% RSLogix 500 project Examen Certificación.RSS, saved by version 9.00.00.04 %
PROJECT "UNTITLED"    % processor: MicroLogix 1200 %

PROGRAM FILES
  LAD 2 "MAIN"  6 rungs
  LAD 3 "ENTRADAS"  6 rungs
  LAD 4 "SALIDAS"  4 rungs
  LAD 5 "MANUAL"  4 rungs
  LAD 6 "AUTOMATICO"  11 rungs
  LAD 7 "PARPADEOS"  5 rungs
  LAD 8 "LS"  2 rungs

DATA FILES
  O0 OUTPUT  4 elements
  I1 INPUT  4 elements
  S2 STATUS  66 elements
  B3 BINARY  4 elements
  T4 TIMER  3 elements
  C5 COUNTER  2 elements
  R6 CONTROL  1 elements
  N7 INTEGER  1 elements
  F8 FLOAT  1 elements

LADDER 2 "MAIN"
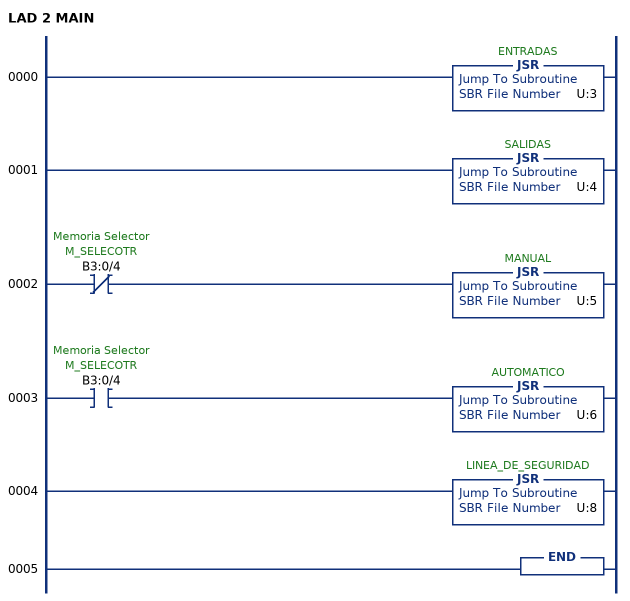
% Rung: 0 %
SOR JSR U:3 EOR
%   U:3  ENTRADAS %
% Rung: 1 %
SOR JSR U:4 EOR
%   U:4  SALIDAS %
% Rung: 2 %
SOR XIO B3:0/4 JSR U:5 EOR
%   B3:0/4  M_SELECOTR  "Memoria Selector" %
%   U:5  MANUAL %
% Rung: 3 %
SOR XIC B3:0/4 JSR U:6 EOR
%   B3:0/4  M_SELECOTR  "Memoria Selector" %
%   U:6  AUTOMATICO %
% Rung: 4 %
SOR JSR U:8 EOR
%   U:8  LINEA_DE_SEGURIDAD %
% Rung: 5 %
SOR END EOR

LADDER 3 "ENTRADAS"
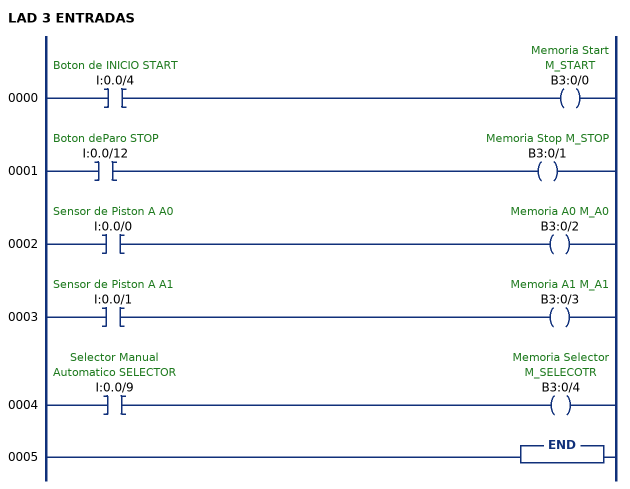
% Rung: 0 %
SOR XIC I:0.0/4 OTE B3:0/0 EOR
%   I:0.0/4  START  "Boton de INICIO" %
%   B3:0/0  M_START  "Memoria Start" %
% Rung: 1 %
SOR XIC I:0.0/12 OTE B3:0/1 EOR
%   I:0.0/12  STOP  "Boton deParo" %
%   B3:0/1  M_STOP  "Memoria Stop" %
% Rung: 2 %
SOR XIC I:0.0/0 OTE B3:0/2 EOR
%   I:0.0/0  A0  "Sensor de Piston A" %
%   B3:0/2  M_A0  "Memoria A0" %
% Rung: 3 %
SOR XIC I:0.0/1 OTE B3:0/3 EOR
%   I:0.0/1  A1  "Sensor de Piston A" %
%   B3:0/3  M_A1  "Memoria A1" %
% Rung: 4 %
SOR XIC I:0.0/9 OTE B3:0/4 EOR
%   I:0.0/9  SELECTOR  "Selector Manual Automatico" %
%   B3:0/4  M_SELECOTR  "Memoria Selector" %
% Rung: 5 %
SOR END EOR

LADDER 4 "SALIDAS"
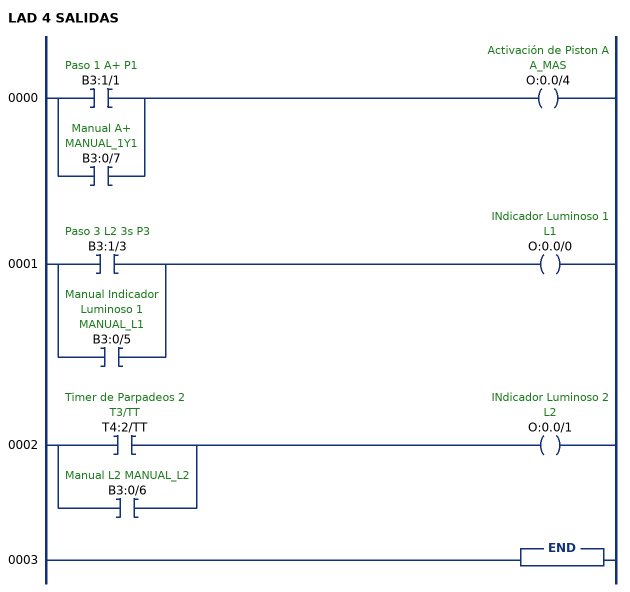
% Rung: 0 %
SOR BST XIC B3:1/1 NXB XIC B3:0/7 BND OTE O:0.0/4 EOR
%   B3:1/1  P1  "Paso 1 A+" %
%   B3:0/7  MANUAL_1Y1  "Manual A+" %
%   O:0.0/4  A_MAS  "Activación de Piston A" %
% Rung: 1 %
SOR BST XIC B3:1/3 NXB XIC B3:0/5 BND OTE O:0.0/0 EOR
%   B3:1/3  P3  "Paso 3 L2 3s" %
%   B3:0/5  MANUAL_L1  "Manual Indicador Luminoso 1" %
%   O:0.0/0  L1  "INdicador Luminoso 1" %
% Rung: 2 %
SOR BST XIC T4:2/TT NXB XIC B3:0/6 BND OTE O:0.0/1 EOR
%   T4:2  T3  "Timer de Parpadeos 2" %
%   B3:0/6  MANUAL_L2  "Manual L2" %
%   O:0.0/1  L2  "INdicador Luminoso 2" %
% Rung: 3 %
SOR END EOR

LADDER 5 "MANUAL"
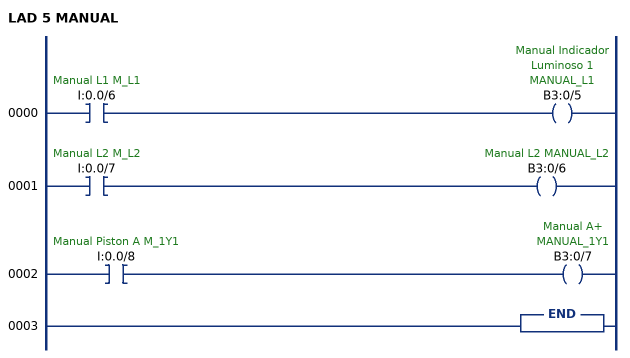
% Rung: 0 %
SOR XIC I:0.0/6 OTE B3:0/5 EOR
%   I:0.0/6  M_L1  "Manual L1" %
%   B3:0/5  MANUAL_L1  "Manual Indicador Luminoso 1" %
% Rung: 1 %
SOR XIC I:0.0/7 OTE B3:0/6 EOR
%   I:0.0/7  M_L2  "Manual L2" %
%   B3:0/6  MANUAL_L2  "Manual L2" %
% Rung: 2 %
SOR XIC I:0.0/8 OTE B3:0/7 EOR
%   I:0.0/8  M_1Y1  "Manual Piston A" %
%   B3:0/7  MANUAL_1Y1  "Manual A+" %
% Rung: 3 %
SOR END EOR

LADDER 6 "AUTOMATICO"
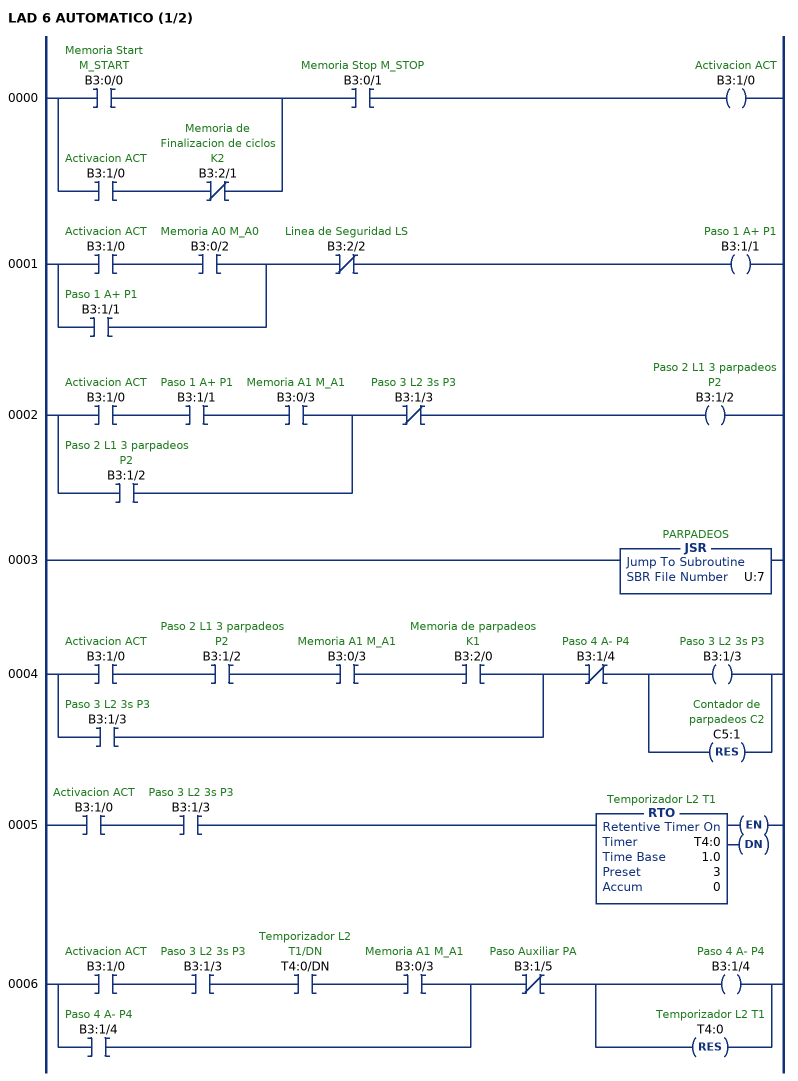
% Rung: 0 %
SOR BST XIC B3:0/0 NXB XIC B3:1/0 XIO B3:2/1 BND XIC B3:0/1 OTE B3:1/0 EOR
%   B3:0/0  M_START  "Memoria Start" %
%   B3:1/0  ACT  "Activacion" %
%   B3:2/1  K2  "Memoria de Finalizacion de ciclos" %
%   B3:0/1  M_STOP  "Memoria Stop" %
% Rung: 1 %
SOR BST XIC B3:1/0 XIC B3:0/2 NXB XIC B3:1/1 BND XIO B3:2/2 OTE B3:1/1 EOR
%   B3:1/0  ACT  "Activacion" %
%   B3:0/2  M_A0  "Memoria A0" %
%   B3:1/1  P1  "Paso 1 A+" %
%   B3:2/2  LS  "Linea de Seguridad" %
% Rung: 2 %
SOR BST XIC B3:1/0 XIC B3:1/1 XIC B3:0/3 NXB XIC B3:1/2 BND XIO B3:1/3 OTE B3:1/2 EOR
%   B3:1/0  ACT  "Activacion" %
%   B3:1/1  P1  "Paso 1 A+" %
%   B3:0/3  M_A1  "Memoria A1" %
%   B3:1/2  P2  "Paso 2 L1 3 parpadeos" %
%   B3:1/3  P3  "Paso 3 L2 3s" %
% Rung: 3 %
SOR JSR U:7 EOR
%   U:7  PARPADEOS %
% Rung: 4 %
SOR BST XIC B3:1/0 XIC B3:1/2 XIC B3:0/3 XIC B3:2/0 NXB XIC B3:1/3 BND XIO B3:1/4 BST OTE B3:1/3 NXB RES C5:1 BND EOR
%   B3:1/0  ACT  "Activacion" %
%   B3:1/2  P2  "Paso 2 L1 3 parpadeos" %
%   B3:0/3  M_A1  "Memoria A1" %
%   B3:2/0  K1  "Memoria de parpadeos" %
%   B3:1/3  P3  "Paso 3 L2 3s" %
%   B3:1/4  P4  "Paso 4 A-" %
%   C5:1  C2  "Contador de parpadeos" %
% Rung: 5 %
SOR XIC B3:1/0 XIC B3:1/3 RTO T4:0 1.0 3 0 EOR
%   B3:1/0  ACT  "Activacion" %
%   B3:1/3  P3  "Paso 3 L2 3s" %
%   T4:0  T1  "Temporizador L2" %
% Rung: 6 %
SOR BST XIC B3:1/0 XIC B3:1/3 XIC T4:0/DN XIC B3:0/3 NXB XIC B3:1/4 BND XIO B3:1/5 BST OTE B3:1/4 NXB RES T4:0 BND EOR
%   B3:1/0  ACT  "Activacion" %
%   B3:1/3  P3  "Paso 3 L2 3s" %
%   T4:0  T1  "Temporizador L2" %
%   B3:0/3  M_A1  "Memoria A1" %
%   B3:1/4  P4  "Paso 4 A-" %
%   B3:1/5  PA  "Paso Auxiliar" %

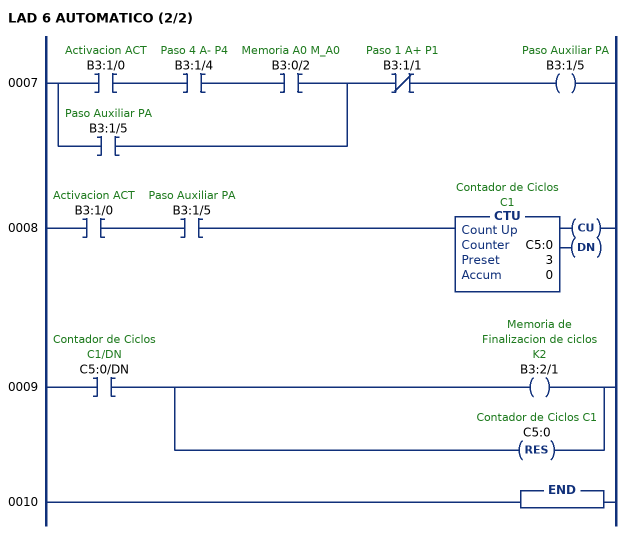
% Rung: 7 %
SOR BST XIC B3:1/0 XIC B3:1/4 XIC B3:0/2 NXB XIC B3:1/5 BND XIO B3:1/1 OTE B3:1/5 EOR
%   B3:1/0  ACT  "Activacion" %
%   B3:1/4  P4  "Paso 4 A-" %
%   B3:0/2  M_A0  "Memoria A0" %
%   B3:1/5  PA  "Paso Auxiliar" %
%   B3:1/1  P1  "Paso 1 A+" %
% Rung: 8 %
SOR XIC B3:1/0 XIC B3:1/5 CTU C5:0 3 0 EOR
%   B3:1/0  ACT  "Activacion" %
%   B3:1/5  PA  "Paso Auxiliar" %
%   C5:0  C1  "Contador de Ciclos" %
% Rung: 9 %
SOR XIC C5:0/DN BST OTE B3:2/1 NXB RES C5:0 BND EOR
%   C5:0  C1  "Contador de Ciclos" %
%   B3:2/1  K2  "Memoria de Finalizacion de ciclos" %
% Rung: 10 %
SOR END EOR

LADDER 7 "PARPADEOS"
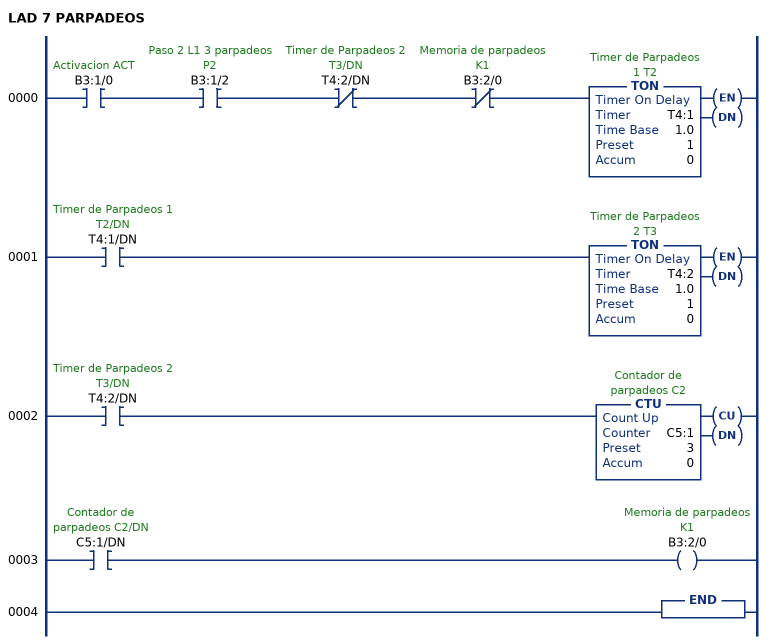
% Rung: 0 %
SOR XIC B3:1/0 XIC B3:1/2 XIO T4:2/DN XIO B3:2/0 TON T4:1 1.0 1 0 EOR
%   B3:1/0  ACT  "Activacion" %
%   B3:1/2  P2  "Paso 2 L1 3 parpadeos" %
%   T4:2  T3  "Timer de Parpadeos 2" %
%   B3:2/0  K1  "Memoria de parpadeos" %
%   T4:1  T2  "Timer de Parpadeos 1" %
% Rung: 1 %
SOR XIC T4:1/DN TON T4:2 1.0 1 0 EOR
%   T4:1  T2  "Timer de Parpadeos 1" %
%   T4:2  T3  "Timer de Parpadeos 2" %
% Rung: 2 %
SOR XIC T4:2/DN CTU C5:1 3 0 EOR
%   T4:2  T3  "Timer de Parpadeos 2" %
%   C5:1  C2  "Contador de parpadeos" %
% Rung: 3 %
SOR XIC C5:1/DN OTE B3:2/0 EOR
%   C5:1  C2  "Contador de parpadeos" %
%   B3:2/0  K1  "Memoria de parpadeos" %
% Rung: 4 %
SOR END EOR

LADDER 8 "LS"
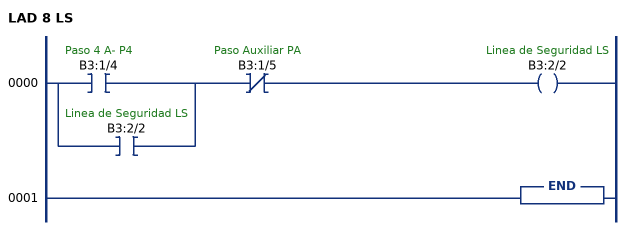
% Rung: 0 %
SOR BST XIC B3:1/4 NXB XIC B3:2/2 BND XIO B3:1/5 OTE B3:2/2 EOR
%   B3:1/4  P4  "Paso 4 A-" %
%   B3:2/2  LS  "Linea de Seguridad" %
%   B3:1/5  PA  "Paso Auxiliar" %
% Rung: 1 %
SOR END EOR

DATA TABLE (non-zero values as saved)
DATA T4
% .PRE .ACC %
% T4:0 % 3 0
% T4:1 % 1 0
% T4:2 % 1 0
DATA C5
% .PRE .ACC %
% C5:0 % 3 0
% C5:1 % 3 0
